// TIA Portal V16 export
// export: Created 2022-11-17T15:49:15.7400397Z, ExportSetting WithDefaults, DisplayName Totally Integrated Automation Portal, DisplayVersion V16 Update 6, DisplayName TIA Portal Version Control Interface, DisplayVersion V16 Update 2, DisplayName TIA Portal Openness, DisplayVersion V16 Update 6, DisplayName SINAMICS Startdrive Advanced, DisplayVersion V16 Update 5, DisplayName SINAMICS Startdrive G130, G150, S120, S150, SINAMICS MV, S210, DisplayVersion V16 Update 5, DisplayName SINAMICS Startdrive G110M, G120, G120C, G120D, G120P, G115D, DisplayVersion V16 Update 5, DisplayName STEP 7 Professional, DisplayVersion V16 Update 6, DisplayName STEP 7 Safety, DisplayVersion V16, DisplayName WinCC Advanced, DisplayVersion V16 Update 6
FUNCTION "FC07_FilmBroken&Test" : Void   // FC7, LAD
TITLE = Film broken or ended management
{ S7_Optimized_Access := 'FALSE' }
AUTHOR : Robopac
VERSION : 0.0
// stored: AutoNumber false, IsIECCheckEnabled false, SetENOAutomatically false, UDAEnableTagReadback false
   VAR_TEMP   // added for the SCL form of the ladder/FBD networks
      _w1 : Bool;
   END_VAR
BEGIN

REGION Network 1: Delay for test cycle
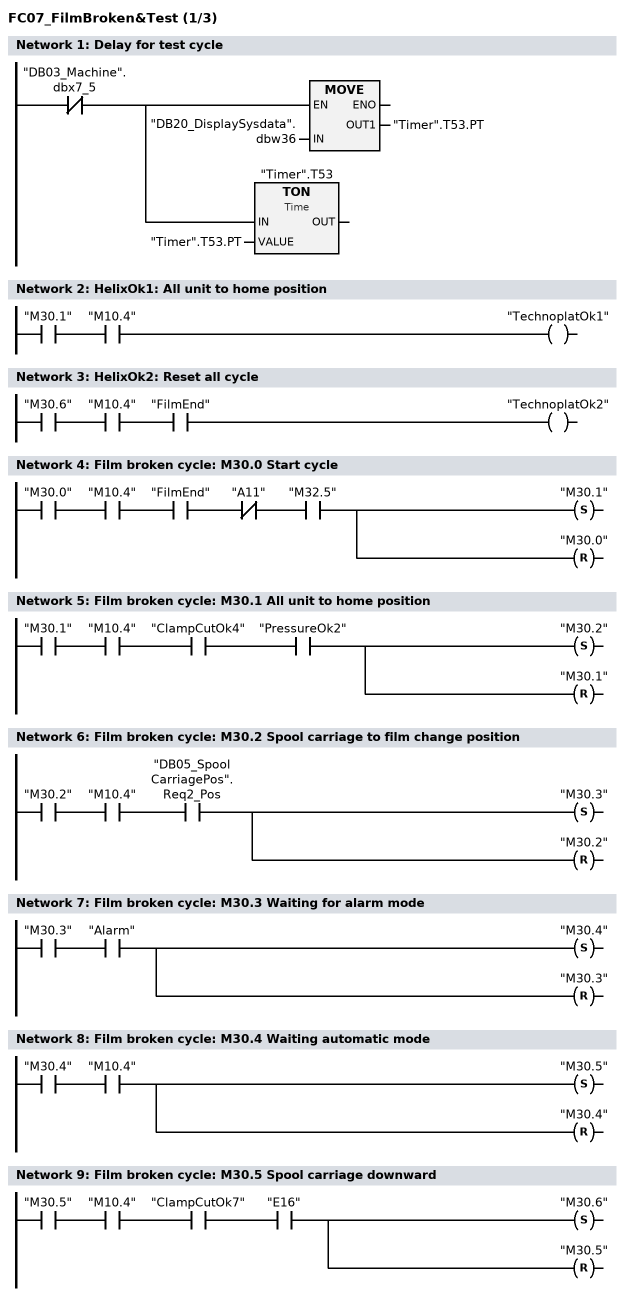
   #_w1 := NOT "DB03_Machine".dbx7_5;
   IF #_w1 THEN "Timer".T53.PT := "DB20_DisplaySysdata".dbw36; END_IF;
   "Timer".T53.TON(IN := #_w1, PT := "Timer".T53.PT);   // TON coil
END_REGION

REGION Network 2: HelixOk1: All unit to home position
   RUNG wire#powerrail
      Contact( "M30.1" )
      Contact( "M10.4" )
      Coil( "TechnoplatOk1" )
   END_RUNG
   // the same network as SCL:
   "TechnoplatOk1" := "M30.1" AND "M10.4";
END_REGION

REGION Network 3: HelixOk2: Reset all cycle
   RUNG wire#powerrail
      Contact( "M30.6" )
      Contact( "M10.4" )
      Contact( "FilmEnd" )
      Coil( "TechnoplatOk2" )
   END_RUNG
   // the same network as SCL:
   "TechnoplatOk2" := "M30.6" AND "M10.4" AND "FilmEnd";
END_REGION

REGION Network 4: Film broken cycle: M30.0 Start cycle
   RUNG wire#powerrail
      Contact( "M30.0" )
      Contact( "M10.4" )
      Contact( "FilmEnd" )
      I_Contact( "A11" )
      Contact( "M32.5" )
      wire#w1
      S_Coil( "M30.1" )
   END_RUNG
   RUNG wire#w1
      R_Coil( "M30.0" )
   END_RUNG
   // the same network as SCL:
   IF "M30.0" AND "M10.4" AND "FilmEnd" AND NOT "A11" AND "M32.5" THEN
       "M30.1" := TRUE;
       "M30.0" := FALSE;
   END_IF;
END_REGION

REGION Network 5: Film broken cycle: M30.1 All unit to home position
   RUNG wire#powerrail
      Contact( "M30.1" )
      Contact( "M10.4" )
      Contact( "ClampCutOk4" )
      Contact( "PressureOk2" )
      wire#w1
      S_Coil( "M30.2" )
   END_RUNG
   RUNG wire#w1
      R_Coil( "M30.1" )
   END_RUNG
   // the same network as SCL:
   IF "M30.1" AND "M10.4" AND "ClampCutOk4" AND "PressureOk2" THEN
       "M30.2" := TRUE;
       "M30.1" := FALSE;
   END_IF;
END_REGION

REGION Network 6: Film broken cycle: M30.2 Spool carriage to film change position
   RUNG wire#powerrail
      Contact( "M30.2" )
      Contact( "M10.4" )
      Contact( "DB05_SpoolCarriagePos".Req2_Pos )
      wire#w1
      S_Coil( "M30.3" )
   END_RUNG
   RUNG wire#w1
      R_Coil( "M30.2" )
   END_RUNG
   // the same network as SCL:
   IF "M30.2" AND "M10.4" AND "DB05_SpoolCarriagePos".Req2_Pos THEN
       "M30.3" := TRUE;
       "M30.2" := FALSE;
   END_IF;
END_REGION

REGION Network 7: Film broken cycle: M30.3 Waiting for alarm mode
   RUNG wire#powerrail
      Contact( "M30.3" )
      Contact( "Alarm" )
      wire#w1
      S_Coil( "M30.4" )
   END_RUNG
   RUNG wire#w1
      R_Coil( "M30.3" )
   END_RUNG
   // the same network as SCL:
   IF "M30.3" AND "Alarm" THEN
       "M30.4" := TRUE;
       "M30.3" := FALSE;
   END_IF;
END_REGION

REGION Network 8: Film broken cycle: M30.4 Waiting automatic mode
   RUNG wire#powerrail
      Contact( "M30.4" )
      Contact( "M10.4" )
      wire#w1
      S_Coil( "M30.5" )
   END_RUNG
   RUNG wire#w1
      R_Coil( "M30.4" )
   END_RUNG
   // the same network as SCL:
   IF "M30.4" AND "M10.4" THEN
       "M30.5" := TRUE;
       "M30.4" := FALSE;
   END_IF;
END_REGION

REGION Network 9: Film broken cycle: M30.5 Spool carriage downward
   RUNG wire#powerrail
      Contact( "M30.5" )
      Contact( "M10.4" )
      Contact( "ClampCutOk7" )
      Contact( "E16" )
      wire#w1
      S_Coil( "M30.6" )
   END_RUNG
   RUNG wire#w1
      R_Coil( "M30.5" )
   END_RUNG
   // the same network as SCL:
   IF "M30.5" AND "M10.4" AND "ClampCutOk7" AND "E16" THEN
       "M30.6" := TRUE;
       "M30.5" := FALSE;
   END_IF;
END_REGION

REGION Network 10: Film broken cycle: M30.6 Waiting step
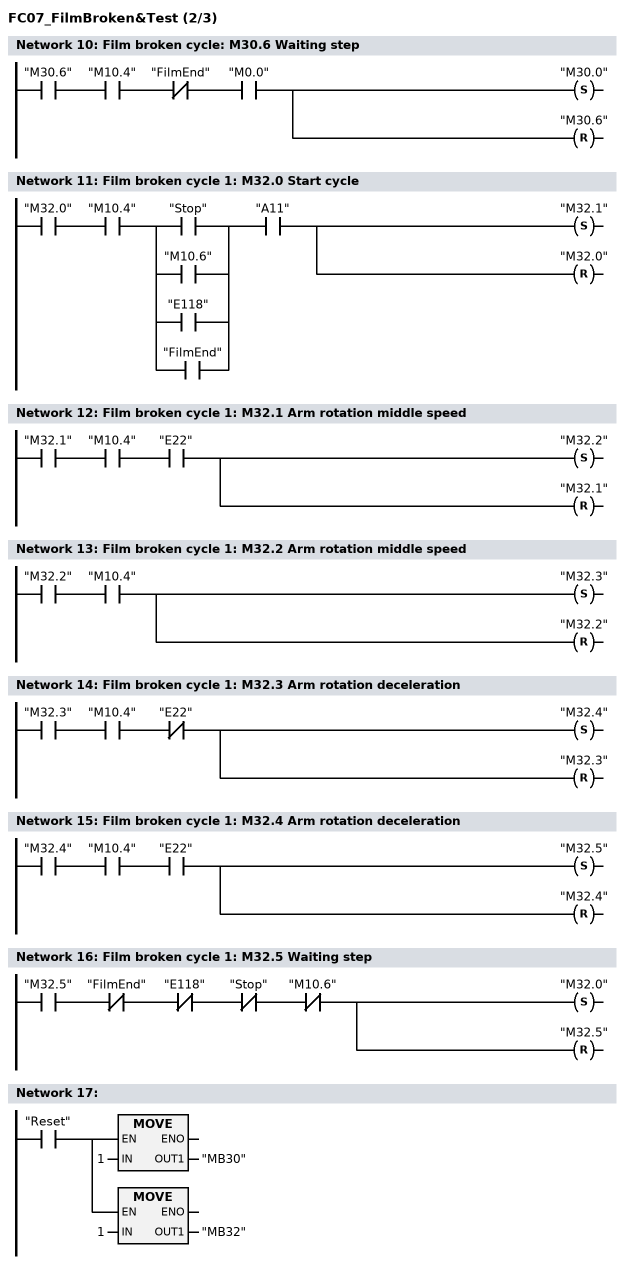
   RUNG wire#powerrail
      Contact( "M30.6" )
      Contact( "M10.4" )
      I_Contact( "FilmEnd" )
      Contact( "M0.0" )
      wire#w1
      S_Coil( "M30.0" )
   END_RUNG
   RUNG wire#w1
      R_Coil( "M30.6" )
   END_RUNG
   // the same network as SCL:
   IF "M30.6" AND "M10.4" AND NOT "FilmEnd" AND "M0.0" THEN
       "M30.0" := TRUE;
       "M30.6" := FALSE;
   END_IF;
END_REGION

REGION Network 11: Film broken cycle 1: M32.0 Start cycle
   RUNG wire#powerrail
      Contact( "M32.0" )
      Contact( "M10.4" )
      wire#w1
      Contact( "Stop" )
      wire#w2
      Contact( "A11" )
      wire#w3
      S_Coil( "M32.1" )
   END_RUNG
   RUNG wire#w1
      Contact( "M10.6" )
   END_RUNG wire#w2
   RUNG wire#w1
      Contact( "E118" )
   END_RUNG wire#w2
   RUNG wire#w1
      Contact( "FilmEnd" )
   END_RUNG wire#w2
   RUNG wire#w3
      R_Coil( "M32.0" )
   END_RUNG
   // the same network as SCL:
   IF "M32.0" AND "M10.4" AND ("Stop" OR "M10.6" OR "E118" OR "FilmEnd") AND "A11" THEN
       "M32.1" := TRUE;
       "M32.0" := FALSE;
   END_IF;
END_REGION

REGION Network 12: Film broken cycle 1: M32.1 Arm rotation middle speed
   RUNG wire#powerrail
      Contact( "M32.1" )
      Contact( "M10.4" )
      Contact( "E22" )
      wire#w1
      S_Coil( "M32.2" )
   END_RUNG
   RUNG wire#w1
      R_Coil( "M32.1" )
   END_RUNG
   // the same network as SCL:
   IF "M32.1" AND "M10.4" AND "E22" THEN
       "M32.2" := TRUE;
       "M32.1" := FALSE;
   END_IF;
END_REGION

REGION Network 13: Film broken cycle 1: M32.2 Arm rotation middle speed
   RUNG wire#powerrail
      Contact( "M32.2" )
      Contact( "M10.4" )
      wire#w1
      S_Coil( "M32.3" )
   END_RUNG
   RUNG wire#w1
      R_Coil( "M32.2" )
   END_RUNG
   // the same network as SCL:
   IF "M32.2" AND "M10.4" THEN
       "M32.3" := TRUE;
       "M32.2" := FALSE;
   END_IF;
END_REGION

REGION Network 14: Film broken cycle 1: M32.3 Arm rotation deceleration
   RUNG wire#powerrail
      Contact( "M32.3" )
      Contact( "M10.4" )
      I_Contact( "E22" )
      wire#w1
      S_Coil( "M32.4" )
   END_RUNG
   RUNG wire#w1
      R_Coil( "M32.3" )
   END_RUNG
   // the same network as SCL:
   IF "M32.3" AND "M10.4" AND NOT "E22" THEN
       "M32.4" := TRUE;
       "M32.3" := FALSE;
   END_IF;
END_REGION

REGION Network 15: Film broken cycle 1: M32.4 Arm rotation deceleration
   RUNG wire#powerrail
      Contact( "M32.4" )
      Contact( "M10.4" )
      Contact( "E22" )
      wire#w1
      S_Coil( "M32.5" )
   END_RUNG
   RUNG wire#w1
      R_Coil( "M32.4" )
   END_RUNG
   // the same network as SCL:
   IF "M32.4" AND "M10.4" AND "E22" THEN
       "M32.5" := TRUE;
       "M32.4" := FALSE;
   END_IF;
END_REGION

REGION Network 16: Film broken cycle 1: M32.5 Waiting step
   RUNG wire#powerrail
      Contact( "M32.5" )
      I_Contact( "FilmEnd" )
      I_Contact( "E118" )
      I_Contact( "Stop" )
      I_Contact( "M10.6" )
      wire#w1
      S_Coil( "M32.0" )
   END_RUNG
   RUNG wire#w1
      R_Coil( "M32.5" )
   END_RUNG
   // the same network as SCL:
   IF "M32.5" AND NOT "FilmEnd" AND NOT "E118" AND NOT "Stop" AND NOT "M10.6" THEN
       "M32.0" := TRUE;
       "M32.5" := FALSE;
   END_IF;
END_REGION

REGION Network 17
   RUNG wire#powerrail
      Contact( "Reset" )
      wire#w1
      { S7_GenerateENO := "TRUE" } Move(in := 1, out1 => "MB30")
   END_RUNG
   RUNG wire#w1
      { S7_GenerateENO := "TRUE" } Move(in := 1, out1 => "MB32")
   END_RUNG
   // the same network as SCL:
   IF "Reset" THEN
       "MB30" := 1;
       "MB32" := 1;
   END_IF;
END_REGION

REGION Network 18: Machine cycle: M1.5 Waiting step
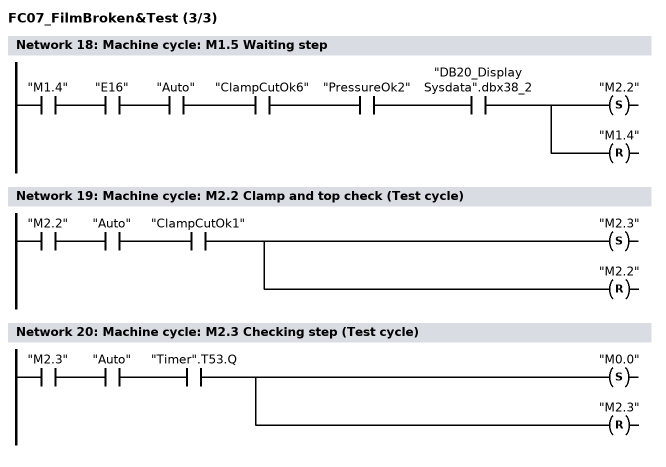
   RUNG wire#powerrail
      Contact( "M1.4" )
      Contact( "E16" )
      Contact( "Auto" )
      Contact( "ClampCutOk6" )
      Contact( "PressureOk2" )
      Contact( "DB20_DisplaySysdata".dbx38_2 )
      wire#w1
      S_Coil( "M2.2" )
   END_RUNG
   RUNG wire#w1
      R_Coil( "M1.4" )
   END_RUNG
   // the same network as SCL:
   IF "M1.4" AND "E16" AND "Auto" AND "ClampCutOk6" AND "PressureOk2" AND "DB20_DisplaySysdata".dbx38_2 THEN
       "M2.2" := TRUE;
       "M1.4" := FALSE;
   END_IF;
END_REGION

REGION Network 19: Machine cycle: M2.2 Clamp and top check (Test cycle)
   RUNG wire#powerrail
      Contact( "M2.2" )
      Contact( "Auto" )
      Contact( "ClampCutOk1" )
      wire#w1
      S_Coil( "M2.3" )
   END_RUNG
   RUNG wire#w1
      R_Coil( "M2.2" )
   END_RUNG
   // the same network as SCL:
   IF "M2.2" AND "Auto" AND "ClampCutOk1" THEN
       "M2.3" := TRUE;
       "M2.2" := FALSE;
   END_IF;
END_REGION

REGION Network 20: Machine cycle: M2.3 Checking step (Test cycle)
   RUNG wire#powerrail
      Contact( "M2.3" )
      Contact( "Auto" )
      Contact( "Timer".T53.Q )
      wire#w1
      S_Coil( "M0.0" )
   END_RUNG
   RUNG wire#w1
      R_Coil( "M2.3" )
   END_RUNG
   // the same network as SCL:
   IF "M2.3" AND "Auto" AND "Timer".T53.Q THEN
       "M0.0" := TRUE;
       "M2.3" := FALSE;
   END_IF;
END_REGION
END_FUNCTION
